// TIA Portal V19 export
DATA_BLOCK "Network_DB"   // DB31
// stored: InstanceOfName Network XC208, InstanceOfType FB
"Network XC208"
   // VAR_INPUT
   //    Trigger : Bool;
   //    HWID : HW_ANY;
   // END_VAR
   // VAR_OUTPUT
   //    Error : Bool;
   //    Status : Word;
   // END_VAR
   // VAR_IN_OUT
   //    NetworkHMI_PortInfo : Variant;
   // END_VAR
   // VAR
   //    PortInformation { S7_SetPoint := 'True'} : "LPNDR_ReadGlobalInfo";
   // END_VAR
BEGIN
END_DATA_BLOCK
